Fanuc KAREL source: f_float_t.kl

PROGRAM F_FLOAT_T
VAR r : REAL
BEGIN
  r = 123.45
  r = 0.1
  r = 1000000.0
  r = 0.000123
  r = 1.0E10
  r = -2.5
  r = 3
END F_FLOAT_T
